# EPICS autosave request: iocBoot/sioc-li11-bl01/blen_manual.req
file "manual.req" AREA=LI11,POS=359,INST=BZ11359A
file "manual.req" AREA=LI11,POS=359,INST=BZ11359B
